# B&R Automation Studio project ShowCase2Mo410Test
Automation Studio 4.10.5.38 SP; technology packages: mapp 5.23.1, mappCockpit 5.23.0, mappMotion 5.23.1, mappView 5.23.0

## Configuration Config1

CPU X20CP1586, AutomationRuntime B4.91, Build 4.1.2, Safety 0.0, Vc 

### Task classes (Cpu.sw)
```
Cyclic#1:
  BoxLift <- BoxLift.prg
  ComTCP_P <- Libraries.ComTCP.ComTCP_P.prg
  AlarmBlink <- AlarmBlink.prg
  Axis1ST <- Axis1ST.prg
Cyclic#4:
  RecipeMgmt <- RecipeMgmt.prg
  PowerON <- PowerON.prg
  CamAutomat <- CamAutomat.prg
  LDMPAccess <- LDMPAccess.prg
DataObjects: McAcpSys
NcDataObjects: Cam <- Cam.dob, McDriveLog
Binaries: TCData, mvLoader, TCLang, udbdef, arsvcreg, mCoWebSc, arflatprv, arcoal, McAcpDrv, McAcpSim, arconfig, asfw, ashwd, iomap, User, Role, sysconf, TC, ashwac, Config_3, Config_2, Config, Config_1, Settings
Libraries: MTBasics, brsystem, MTTypes, sys_lib, runtime, ComTCP_L, operator, astime, AsTCP, standard, AsArLog, AsBrStr, MpRecipe, MpBase, McBase, CoTrace, AsZip, FileIO, MpAxis, McAxis, McAcpAx, asieccon, arssl, asepl, powerlnk
```

### Hardware
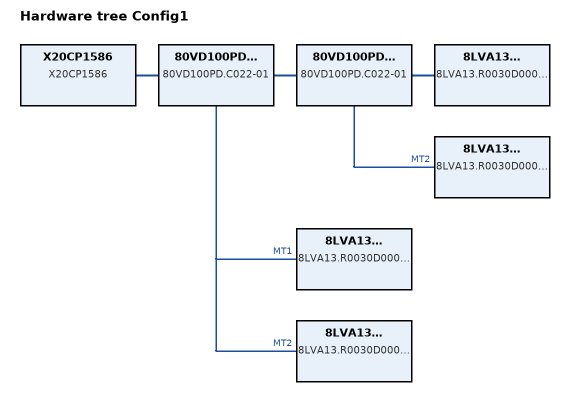
```
80VD100PD.C022-01 : 80VD100PD.C022-01 v2.5.0.0  [PLK1 -> X20CP1586.IF3 (NodeNumber=2) [Cable Type=PowerlinkCable, Length=10, Version=1.0.0.3]; PLK2 -> 80VD100PD.C022-01a.PLK1 (NodeNumber=2) [Cable Type=PowerlinkCable, Length=10, Version=1.0.0.3]; MT2 -> 8LVA13.R0030D000-0a.MT]
  DriveConfiguration/Module:
    McAcoposTypeID = AcoposMicroDConfig
    ActivateACOPOSSimulationOnPLC = 0
  DriveConfiguration/Encoder/EncoderX6A/InterfaceType:
    ResolverPolepairs = 1
  DriveConfiguration/Encoder/EncoderX6B/InterfaceType:
    ResolverPolepairs = 1
  DriveConfiguration/Channel[1]/RealAxis:
    AxisReference = gAxis3_MpLink
    MechanicalElementsIsInvisible = 0
  DriveConfiguration/Channel[1]/RealAxis/MechanicalElements/Gearbox:
    InputIsReadOnly = 0
    Input = 1
    OutputIsReadOnly = 0
    Output = 1
  DriveConfiguration/Channel[1]/RealAxis/MechanicalElements/RotaryToLinearTransformation:
    ReferenceDistanceIsReadOnly = 0
    ReferenceDistance = 1
  DriveConfiguration/Channel[1]/RealAxis/Controller:
    ModeIsReadOnly = 0
    Mode = PositionController
  DriveConfiguration/Channel[1]/RealAxis/Controller/Mode/Position:
    ProportionalGain = 50.0
    IntegrationTime = 0.0
    PredictionTime = 0.0004
    TotalDelayTime = 0.0004
  DriveConfiguration/Channel[1]/RealAxis/Controller/Mode/Speed:
    ProportionalGainIsReadOnly = 0
    ProportionalGain = 2.0
    IntegrationTimeIsReadOnly = 0
    IntegrationTime = 0.0
    FilterTimeIsReadOnly = 0
    FilterTime = 0.0
  DriveConfiguration/Channel[1]/RealAxis/Controller/Mode/LoopFilters:
    LoopFilterXIsReadOnly = 0
    LoopFilter1 = NotUsed
    LoopFilter2 = NotUsed
    LoopFilter3 = NotUsed
  DriveConfiguration/Channel[1]/RealAxis/Homing:
    ModeIsReadOnly = 0
    Mode = Direct
  DriveConfiguration/Channel[1]/RealAxis/Homing/Mode:
    Position = 0.0
    ReferencePulse = NotUsed
  DriveConfiguration/Channel[1]/RealAxis/Homing:
    RestorePositionVariable = 
  DriveConfiguration/Channel[1]/RealAxis/StopReaction:
    QuickstopIsReadOnly = 0
    Quickstop = DecelerationLimit
    DriveErrorIsReadOnly = 0
    DriveError = DecelerationLimit
  DriveConfiguration/Channel[1]/RealAxis/MovementErrorLimits:
    PositionError = 300
    VelocityErrorMonitoring = Automatic1
  DriveConfiguration/Channel[1]/RealAxis:
    JerkFilterIsReadOnly = 0
    JerkFilter = NotUsed
    ZeroVibrationFilter = NotUsed
  DriveConfiguration/Channel[1]/RealAxis/DigitalInputs/HomingSwitch:
    SourceIsReadOnly = 0
    Source = NotUsed
    Level = High
  DriveConfiguration/Channel[1]/RealAxis/DigitalInputs/PositiveLimitSwitch:
    SourceIsReadOnly = 0
    Source = NotUsed
    Level = High
  DriveConfiguration/Channel[1]/RealAxis/DigitalInputs/NegativeLimitSwitch:
    SourceIsReadOnly = 0
    Source = NotUsed
    Level = High
  DriveConfiguration/Channel[1]/RealAxis/DigitalInputs/Trigger1:
    Source = X2Trigger1
    Level = High
  DriveConfiguration/Channel[1]/RealAxis/DigitalInputs/Trigger2:
    Source = X2Trigger2
    Level = High
  DriveConfiguration/Channel[1]/RealAxis/DigitalInputs/Quickstop:
    Input = NotUsed
  DriveConfiguration/Channel[1]/RealAxis/Simulation:
    SimulationModeOnPLC = SetValueGeneration
    SimulationModeOnACOPOS = NotUsed
  DriveConfiguration/Channel[1]/RealAxis/AxisFeatures:
    FeatureRef[1] = 
  DriveConfiguration/Channel[1]:
    VirtualAxis = Used
  DriveConfiguration/Channel[1]/VirtualAxis:
    AxisReference = gAxisV3_MpLink
  DriveConfiguration/Channel[1]/VirtualAxis/Homing:
    Mode = Direct
  DriveConfiguration/Channel[1]/VirtualAxis/Homing/Mode:
    Position = 0.0
  DriveConfiguration/Channel[1]/VirtualAxis/Homing:
    RestorePositionVariable = 
  DriveConfiguration/Channel[1]/VirtualAxis:
    JerkFilterIsReadOnly = 0
    JerkFilter = NotUsed
    ZeroVibrationFilter = NotUsed
  DriveConfiguration/Channel[1]/ChannelFeatures:
    FeatureRef[1] = Feature_CamList
  DriveConfiguration/Channel[2]/RealAxis:
    AxisReference = gAxis4_MpLink
    MechanicalElementsIsInvisible = 0
  DriveConfiguration/Channel[2]/RealAxis/MechanicalElements/Gearbox:
    InputIsReadOnly = 0
    Input = 1
    OutputIsReadOnly = 0
    Output = 1
  DriveConfiguration/Channel[2]/RealAxis/MechanicalElements/RotaryToLinearTransformation:
    ReferenceDistanceIsReadOnly = 0
    ReferenceDistance = 1
  DriveConfiguration/Channel[2]/RealAxis/Controller:
    ModeIsReadOnly = 0
    Mode = PositionController
  DriveConfiguration/Channel[2]/RealAxis/Controller/Mode/Position:
    ProportionalGain = 50.0
    IntegrationTime = 0.0
    PredictionTime = 0.0004
    TotalDelayTime = 0.0004
  DriveConfiguration/Channel[2]/RealAxis/Controller/Mode/Speed:
    ProportionalGainIsReadOnly = 0
    ProportionalGain = 2.0
    IntegrationTimeIsReadOnly = 0
    IntegrationTime = 0.0
    FilterTimeIsReadOnly = 0
    FilterTime = 0.0
  DriveConfiguration/Channel[2]/RealAxis/Controller/Mode/LoopFilters:
    LoopFilterXIsReadOnly = 0
    LoopFilter1 = NotUsed
    LoopFilter2 = NotUsed
    LoopFilter3 = NotUsed
  DriveConfiguration/Channel[2]/RealAxis/Homing:
    ModeIsReadOnly = 0
    Mode = Direct
  DriveConfiguration/Channel[2]/RealAxis/Homing/Mode:
    Position = 0.0
    ReferencePulse = NotUsed
  DriveConfiguration/Channel[2]/RealAxis/Homing:
    RestorePositionVariable = 
  DriveConfiguration/Channel[2]/RealAxis/StopReaction:
    QuickstopIsReadOnly = 0
    Quickstop = DecelerationLimit
    DriveErrorIsReadOnly = 0
    DriveError = DecelerationLimit
  DriveConfiguration/Channel[2]/RealAxis/MovementErrorLimits:
    PositionError = 300
    VelocityErrorMonitoring = Automatic1
  DriveConfiguration/Channel[2]/RealAxis:
    JerkFilterIsReadOnly = 0
    JerkFilter = NotUsed
    ZeroVibrationFilter = NotUsed
  DriveConfiguration/Channel[2]/RealAxis/DigitalInputs/HomingSwitch:
    SourceIsReadOnly = 0
    Source = NotUsed
    Level = High
  DriveConfiguration/Channel[2]/RealAxis/DigitalInputs/PositiveLimitSwitch:
    SourceIsReadOnly = 0
    Source = NotUsed
    Level = High
  DriveConfiguration/Channel[2]/RealAxis/DigitalInputs/NegativeLimitSwitch:
    SourceIsReadOnly = 0
    Source = NotUsed
    Level = High
  DriveConfiguration/Channel[2]/RealAxis/DigitalInputs/Trigger1:
    Source = X2Trigger1
    Level = High
  DriveConfiguration/Channel[2]/RealAxis/DigitalInputs/Trigger2:
    Source = X2Trigger2
    Level = High
  DriveConfiguration/Channel[2]/RealAxis/DigitalInputs/Quickstop:
    Input = NotUsed
  DriveConfiguration/Channel[2]/RealAxis/Simulation:
    SimulationModeOnPLC = SetValueGeneration
    SimulationModeOnACOPOS = NotUsed
80VD100PD.C022-01a : 80VD100PD.C022-01 v2.5.0.0  [PLK1 -> 80VD100PD.C022-01.PLK2 (NodeNumber=1) [Cable Type=PowerlinkCable, Length=10, Version=1.0.0.3]; MT2 -> 8LVA13.R0030D000-0c.MT]
  DriveConfiguration/Module:
    McAcoposTypeID = AcoposMicroDConfig
    ActivateACOPOSSimulationOnPLC = 0
  DriveConfiguration/Encoder/EncoderX6A/InterfaceType:
    ResolverPolepairs = 1
  DriveConfiguration/Encoder/EncoderX6B/InterfaceType:
    ResolverPolepairs = 1
  DriveConfiguration/Channel[1]/RealAxis:
    AxisReference = gAxis1_MpLink
    MechanicalElementsIsInvisible = 0
  DriveConfiguration/Channel[1]/RealAxis/MechanicalElements/Gearbox:
    InputIsReadOnly = 0
    Input = 1
    OutputIsReadOnly = 0
    Output = 1
  DriveConfiguration/Channel[1]/RealAxis/MechanicalElements/RotaryToLinearTransformation:
    ReferenceDistanceIsReadOnly = 0
    ReferenceDistance = 1
  DriveConfiguration/Channel[1]/RealAxis/Controller:
    ModeIsReadOnly = 0
    Mode = PositionController
  DriveConfiguration/Channel[1]/RealAxis/Controller/Mode/Position:
    ProportionalGain = 50.0
    IntegrationTime = 0.0
    PredictionTime = 0.0004
    TotalDelayTime = 0.0004
  DriveConfiguration/Channel[1]/RealAxis/Controller/Mode/Speed:
    ProportionalGainIsReadOnly = 0
    ProportionalGain = 2.0
    IntegrationTimeIsReadOnly = 0
    IntegrationTime = 0.0
    FilterTimeIsReadOnly = 0
    FilterTime = 0.0
  DriveConfiguration/Channel[1]/RealAxis/Controller/Mode/LoopFilters:
    LoopFilterXIsReadOnly = 0
    LoopFilter1 = NotUsed
    LoopFilter2 = NotUsed
    LoopFilter3 = NotUsed
  DriveConfiguration/Channel[1]/RealAxis/Homing:
    ModeIsReadOnly = 0
    Mode = Direct
  DriveConfiguration/Channel[1]/RealAxis/Homing/Mode:
    Position = 0.0
    ReferencePulse = NotUsed
  DriveConfiguration/Channel[1]/RealAxis/Homing:
    RestorePositionVariable = 
  DriveConfiguration/Channel[1]/RealAxis/StopReaction:
    QuickstopIsReadOnly = 0
    Quickstop = DecelerationLimit
    DriveErrorIsReadOnly = 0
    DriveError = DecelerationLimit
  DriveConfiguration/Channel[1]/RealAxis/MovementErrorLimits:
    PositionError = 300
    VelocityErrorMonitoring = Automatic1
  DriveConfiguration/Channel[1]/RealAxis:
    JerkFilterIsReadOnly = 0
    JerkFilter = NotUsed
    ZeroVibrationFilter = NotUsed
  DriveConfiguration/Channel[1]/RealAxis/DigitalInputs/HomingSwitch:
    SourceIsReadOnly = 0
    Source = NotUsed
    Level = High
  DriveConfiguration/Channel[1]/RealAxis/DigitalInputs/PositiveLimitSwitch:
    SourceIsReadOnly = 0
    Source = NotUsed
    Level = High
  DriveConfiguration/Channel[1]/RealAxis/DigitalInputs/NegativeLimitSwitch:
    SourceIsReadOnly = 0
    Source = NotUsed
    Level = High
  DriveConfiguration/Channel[1]/RealAxis/DigitalInputs/Trigger1:
    Source = X2Trigger1
    Level = High
  DriveConfiguration/Channel[1]/RealAxis/DigitalInputs/Trigger2:
    Source = X2Trigger2
    Level = High
  DriveConfiguration/Channel[1]/RealAxis/DigitalInputs/Quickstop:
    Input = NotUsed
  DriveConfiguration/Channel[1]/RealAxis/Simulation:
    SimulationModeOnPLC = SetValueGeneration
    SimulationModeOnACOPOS = NotUsed
  DriveConfiguration/Channel[1]/RealAxis/AxisFeatures:
    FeatureRef[1] = 
  DriveConfiguration/Channel[1]:
    VirtualAxis = Used
  DriveConfiguration/Channel[1]/VirtualAxis:
    AxisReference = gAxisV_MpLink
  DriveConfiguration/Channel[1]/VirtualAxis/Homing:
    Mode = Direct
  DriveConfiguration/Channel[1]/VirtualAxis/Homing/Mode:
    Position = 0.0
  DriveConfiguration/Channel[1]/VirtualAxis/Homing:
    RestorePositionVariable = 
  DriveConfiguration/Channel[1]/VirtualAxis:
    JerkFilterIsReadOnly = 0
    JerkFilter = NotUsed
    ZeroVibrationFilter = NotUsed
  DriveConfiguration/Channel[1]/ChannelFeatures:
    FeatureRef[1] = Feature_CamList
  DriveConfiguration/Channel[2]/RealAxis:
    AxisReference = gAxis2_MpLink
    MechanicalElementsIsInvisible = 0
  DriveConfiguration/Channel[2]/RealAxis/MechanicalElements/Gearbox:
    InputIsReadOnly = 0
    Input = 1
    OutputIsReadOnly = 0
    Output = 1
  DriveConfiguration/Channel[2]/RealAxis/MechanicalElements/RotaryToLinearTransformation:
    ReferenceDistanceIsReadOnly = 0
    ReferenceDistance = 1
  DriveConfiguration/Channel[2]/RealAxis/Controller:
    ModeIsReadOnly = 0
    Mode = PositionController
  DriveConfiguration/Channel[2]/RealAxis/Controller/Mode/Position:
    ProportionalGain = 50.0
    IntegrationTime = 0.0
    PredictionTime = 0.0004
    TotalDelayTime = 0.0004
  DriveConfiguration/Channel[2]/RealAxis/Controller/Mode/Speed:
    ProportionalGainIsReadOnly = 0
    ProportionalGain = 2.0
    IntegrationTimeIsReadOnly = 0
    IntegrationTime = 0.0
    FilterTimeIsReadOnly = 0
    FilterTime = 0.0
  DriveConfiguration/Channel[2]/RealAxis/Controller/Mode/LoopFilters:
    LoopFilterXIsReadOnly = 0
    LoopFilter1 = NotUsed
    LoopFilter2 = NotUsed
    LoopFilter3 = NotUsed
  DriveConfiguration/Channel[2]/RealAxis/Homing:
    ModeIsReadOnly = 0
    Mode = Direct
  DriveConfiguration/Channel[2]/RealAxis/Homing/Mode:
    Position = 0.0
    ReferencePulse = NotUsed
  DriveConfiguration/Channel[2]/RealAxis/Homing:
    RestorePositionVariable = 
  DriveConfiguration/Channel[2]/RealAxis/StopReaction:
    QuickstopIsReadOnly = 0
    Quickstop = DecelerationLimit
    DriveErrorIsReadOnly = 0
    DriveError = DecelerationLimit
  DriveConfiguration/Channel[2]/RealAxis/MovementErrorLimits:
    PositionError = 300
    VelocityErrorMonitoring = Automatic1
  DriveConfiguration/Channel[2]/RealAxis:
    JerkFilterIsReadOnly = 0
    JerkFilter = NotUsed
    ZeroVibrationFilter = NotUsed
  DriveConfiguration/Channel[2]/RealAxis/DigitalInputs/HomingSwitch:
    SourceIsReadOnly = 0
    Source = NotUsed
    Level = High
  DriveConfiguration/Channel[2]/RealAxis/DigitalInputs/PositiveLimitSwitch:
    SourceIsReadOnly = 0
    Source = NotUsed
    Level = High
  DriveConfiguration/Channel[2]/RealAxis/DigitalInputs/NegativeLimitSwitch:
    SourceIsReadOnly = 0
    Source = NotUsed
    Level = High
  DriveConfiguration/Channel[2]/RealAxis/DigitalInputs/Trigger1:
    Source = X2Trigger1
    Level = High
  DriveConfiguration/Channel[2]/RealAxis/DigitalInputs/Trigger2:
    Source = X2Trigger2
    Level = High
  DriveConfiguration/Channel[2]/RealAxis/DigitalInputs/Quickstop:
    Input = NotUsed
  DriveConfiguration/Channel[2]/RealAxis/Simulation:
    SimulationModeOnPLC = SetValueGeneration
    SimulationModeOnACOPOS = NotUsed
8LVA13.R0030D000-0 : 8LVA13.R0030D000-0 v2.2.0.3  [MT -> 80VD100PD.C022-01.MT1]
  M1/MotorParameters:
    MOTOR_AMB_TEMP_RATED = 40
8LVA13.R0030D000-0a : 8LVA13.R0030D000-0 v2.2.0.3  [MT -> 80VD100PD.C022-01.MT2]
  M1/MotorParameters:
    MOTOR_AMB_TEMP_RATED = 40
8LVA13.R0030D000-0b : 8LVA13.R0030D000-0 v2.2.0.3  [MT -> 80VD100PD.C022-01a.MT1]
  M1/MotorParameters:
    MOTOR_AMB_TEMP_RATED = 40
8LVA13.R0030D000-0c : 8LVA13.R0030D000-0 v2.2.0.3  [MT -> 80VD100PD.C022-01a.MT2]
  M1/MotorParameters:
    MOTOR_AMB_TEMP_RATED = 40
X20CP1586 : X20CP1586 v1.9.0.0
  Connector IF2:
    ActivateDevice = 1
    HostName = mo
    Mode = Manual
    InternetAddress = 192.168.2.32
    SubnetMask = 255.255.255.0
  Connector IF3:
    DNAConfiguration = manual
  ConfigurationID = mappViewGettingStarted_ETA210_T50
  UserPartitionSize = 200
  Simulation = 1
  FileDevice1
  FileDeviceName1 = CSV_Recipes
  FileDevicePath1 = F:\Recipes
  FileDevice2
  FileDeviceName2 = SIM_Recipes
  FileDevicePath2 = C:\Basic
  FtpUser1
  FtpUsername1 = academy
  FtpUserPassword1 = PTbbKbjlQWNQQLeLnvYxsprPr7USEpMWmZovrSfugvI=
  FtpUserSalt1 = LwThsYzd
  FTPAccessRight1 = 0
  ActivateOpcUa = 1
  OpcUaInformationModels_PV_Version = 1
```

### PvMap.vvm - X20CP1586/PvMap.vvm
```iecst
VAR_CONFIG
	::ComTCP_SimActive AT %Q.::gComTCPSimActive; (*Insert your comment here...*)
	::BoxLift:aoBottomBoxReleaseTime AT %Q.::ComTCP_SimOutputs.BottomBox_ReleaseTime; (*Insert your comment here...*)
	::BoxLift:aoTopBoxReleaseTime AT %Q.::ComTCP_SimOutputs.TopBox_ReleaseTime; (*Insert your comment here...*)
	::ComTCP_SimInputs.diConvTop AT %Q.::BoxLift:diConvTop; (*Insert your comment here...*)
	::ComTCP_SimInputs.diConvBottom AT %Q.::BoxLift:diConvBottom; (*Insert your comment here...*)
	::ComTCP_SimInputs.diBoxLift AT %Q.::BoxLift:diBoxLift; (*Insert your comment here...*)
	::ComTCP_SimInputs.diUnloaded AT %Q.::BoxLift:diUnloaded; (*Insert your comment here...*)
	::ComTCP_SimInputs.diLiftTop AT %Q.::BoxLift:diLiftTop; (*Insert your comment here...*)
	::ComTCP_SimInputs.diLiftBottom AT %Q.::BoxLift:diLiftBottom; (*Insert your comment here...*)
	::ComTCP_SimInputs.diLiftUnload AT %Q.::BoxLift:diLiftUnload; (*Insert your comment here...*)
	::BoxLift:doConvTop AT %Q.::ComTCP_SimOutputs.doConvTop; (*Insert your comment here...*)
	::BoxLift:doConvBottom AT %Q.::ComTCP_SimOutputs.doConvBottom; (*Insert your comment here...*)
	::BoxLift:doConvLift AT %Q.::ComTCP_SimOutputs.doConvLift; (*Insert your comment here...*)
	::BoxLift:doLiftTop AT %Q.::ComTCP_SimOutputs.doLiftTop; (*Insert your comment here...*)
	::BoxLift:doLiftBottom AT %Q.::ComTCP_SimOutputs.doLiftBottom; (*Insert your comment here...*)
	::BoxLift:doLiftUnload AT %Q.::ComTCP_SimOutputs.doLiftUnload; (*Insert your comment here...*)
	::BoxLift:aoConvBottomVelocity AT %Q.::ComTCP_SimOutputs.ConvBottom_Velocity; (*Insert your comment here...*)
	::BoxLift:aoConvLiftVelocity AT %Q.::ComTCP_SimOutputs.ConvLift_Velocity; (*Insert your comment here...*)
	::BoxLift:aoConvTopVelocity AT %Q.::ComTCP_SimOutputs.ConvTop_Velocity; (*Insert your comment here...*)
	::BoxLift:aoInfeedConvBottomVelocity AT %Q.::ComTCP_SimOutputs.InfeedConvBottom_Velocity; (*Insert your comment here...*)
	::BoxLift:aoInfeedConvTopVelocity AT %Q.::ComTCP_SimOutputs.InfeedConvTop_Velocity; (*Insert your comment here...*)
	::BoxLift:aoOutfeedConvVelocity AT %Q.::ComTCP_SimOutputs.OutfeedConv_Velocity; (*Insert your comment here...*)
END_VAR
```

### Config_1.axis - X20CP1586/mappMotion/Config_1.axis
```
Element gAxis2_MpLink (Type=axis)  // Axis 2 not used
  BaseTypeIsReadOnly = 0
  BaseType = Linear
    MeasurementUnit = 5066068
    MeasurementResolutionIsReadOnly = 0
    MeasurementResolution = 0.01
    CountDirectionIsReadOnly = 0
    CountDirection = Standard
  MovementLimitsIsReadOnly = 0
  MovementLimits = Internal
    Position:
      LowerLimitMin = -1.79769313486231E308
      UpperLimitMax = 1.79769313486231E308
      LowerLimit = -1000.0
      UpperLimit = 1000.0
    VelocityIsReadOnly = 0
    Velocity:
      VelocityMax = 3.4E38
      Velocity = 15000
    AccelerationIsReadOnly = 0
    Acceleration:
      AccelerationMax = 3.4E38
      Acceleration = 150000
    DecelerationIsReadOnly = 0
    Deceleration:
      DecelerationMax = 3.4E38
      Deceleration = 150000
  Alarms = MpAlarmX
Element gAxisV3_MpLink (Type=axis)  // Virtual axis for servo 3
  BaseTypeIsReadOnly = 0
  BaseType = Linear
    MeasurementUnit = 5066068
    MeasurementResolutionIsReadOnly = 0
    MeasurementResolution = 0.01
    CountDirectionIsReadOnly = 0
    CountDirection = Standard
  MovementLimitsIsReadOnly = 0
  MovementLimits = Internal
    Position:
      LowerLimitMin = -1.79769313486231E308
      UpperLimitMax = 1.79769313486231E308
      LowerLimit = -1000.0
      UpperLimit = 1000.0
    VelocityIsReadOnly = 0
    Velocity:
      VelocityMax = 3.4E38
      Velocity = 15000
    AccelerationIsReadOnly = 0
    Acceleration:
      AccelerationMax = 3.4E38
      Acceleration = 150000
    DecelerationIsReadOnly = 0
    Deceleration:
      DecelerationMax = 3.4E38
      Deceleration = 150000
  Alarms = MpAlarmX
Element gAxisV_MpLink (Type=axis)  // Virtual axis for servo 1
  BaseTypeIsReadOnly = 0
  BaseType = Linear
    MeasurementUnit = 5066068
    MeasurementResolutionIsReadOnly = 0
    MeasurementResolution = 0.01
    CountDirectionIsReadOnly = 0
    CountDirection = Standard
  MovementLimitsIsReadOnly = 0
  MovementLimits = Internal
    Position:
      LowerLimitMin = -1.79769313486231E308
      UpperLimitMax = 1.79769313486231E308
      LowerLimit = -1000.0
      UpperLimit = 1000.0
    VelocityIsReadOnly = 0
    Velocity:
      VelocityMax = 3.4E38
      Velocity = 15000
    AccelerationIsReadOnly = 0
    Acceleration:
      AccelerationMax = 3.4E38
      Acceleration = 150000
    DecelerationIsReadOnly = 0
    Deceleration:
      DecelerationMax = 3.4E38
      Deceleration = 150000
  Alarms = MpAlarmX
Element gAxis4_MpLink (Type=axis)  // Axis 4 not used
  BaseTypeIsReadOnly = 0
  BaseType = Linear
    MeasurementUnit = 5066068
    MeasurementResolutionIsReadOnly = 0
    MeasurementResolution = 0.01
    CountDirectionIsReadOnly = 0
    CountDirection = Standard
  MovementLimitsIsReadOnly = 0
  MovementLimits = Internal
    Position:
      LowerLimitMin = -1.79769313486231E308
      UpperLimitMax = 1.79769313486231E308
      LowerLimit = -1000.0
      UpperLimit = 1000.0
    VelocityIsReadOnly = 0
    Velocity:
      VelocityMax = 3.4E38
      Velocity = 15000
    AccelerationIsReadOnly = 0
    Acceleration:
      AccelerationMax = 3.4E38
      Acceleration = 150000
    DecelerationIsReadOnly = 0
    Deceleration:
      DecelerationMax = 3.4E38
      Deceleration = 150000
  Alarms = MpAlarmX
Element gAxis3_MpLink (Type=axis)  // Axis 3 the lift conveyor with cam automat
  BaseTypeIsReadOnly = 0
  BaseType = Linear
    MeasurementUnit = 5066068
    MeasurementResolutionIsReadOnly = 0
    MeasurementResolution = 0.01
    CountDirectionIsReadOnly = 0
    CountDirection = Standard
  MovementLimitsIsReadOnly = 0
  MovementLimits = Internal
    Position:
      LowerLimitMin = -1.79769313486231E308
      UpperLimitMax = 1.79769313486231E308
      LowerLimit = -1000.0
      UpperLimit = 1000.0
    VelocityIsReadOnly = 0
    Velocity:
      VelocityMax = 3.4E38
      Velocity = 15000
    AccelerationIsReadOnly = 0
    Acceleration:
      AccelerationMax = 3.4E38
      Acceleration = 150000
    DecelerationIsReadOnly = 0
    Deceleration:
      DecelerationMax = 3.4E38
      Deceleration = 150000
  Alarms = MpAlarmX
Element gAxis1_MpLink (Type=axis)  // Axis 1 the lift conveyor
  BaseTypeIsReadOnly = 0
  BaseType = Linear
    MeasurementUnit = 5066068
    MeasurementResolutionIsReadOnly = 0
    MeasurementResolution = 0.01
    CountDirectionIsReadOnly = 0
    CountDirection = Standard
  MovementLimitsIsReadOnly = 0
  MovementLimits = Internal
    Position:
      LowerLimitMin = -1.79769313486231E308
      UpperLimitMax = 1.79769313486231E308
      LowerLimit = -1000.0
      UpperLimit = 1000.0
    VelocityIsReadOnly = 0
    Velocity:
      VelocityMax = 3.4E38
      Velocity = 15000
    AccelerationIsReadOnly = 0
    Acceleration:
      AccelerationMax = 3.4E38
      Acceleration = 150000
    DecelerationIsReadOnly = 0
    Deceleration:
      DecelerationMax = 3.4E38
      Deceleration = 150000
  Alarms = MpAlarmX
```

### Config_3.axisfeature - X20CP1586/mappMotion/Config_3.axisfeature
```
Element Feature_CamList_3 (Type=axisfeature)
  Type = CamList
    CamListRef = CamList_3
Element Feature_CamList (Type=axisfeature)
  Type = CamList
    CamListRef = CamList_1
```

### Config_4.camlist - X20CP1586/mappMotion/Config_4.camlist
```
Element CamList_3 (Type=camlist)
  Row[1]:
    CamName = Cam3
    CamID = 3
    Description
```

## Logical view

Binary libraries used (declarations not repeated): operator, runtime, astime, AsIecCon, brsystem, sys_lib, AsTCP, standard, AsArLog, AsBrStr, MpRecipe, MpBase, McBase, MTBasics 5.12.0, MTTypes, CoTrace, AsZip, FileIO, MpAxis, McAxis, McAcpAx

### Global.typ - Global data types
```iecst
TYPE
	iPhysicParam_typ : 	STRUCT
		UserOutfeedConvVelocity : REAL := 1.0; (*OutfeedConv Velocity Speed ref*)
		UserInfeedConvTopVelocity : REAL := 0.6; (* InfeedConvTop Velocity Speed ref*)
		UserInfeedConvBottomVelocity : REAL := 0.5; (*InfeedConvBottom Velocity Speed ref*)
		UserConvTopVelocity : REAL := 1.0; (* ConvTop VelocitySpeed ref*)
		UserConvLiftVelocity : REAL := 1.0; (* ConvLift Velocity Speed ref*)
		UserConvBottomVelocity : REAL := 1.0; (* Conv Bottom Velocity Speed ref*)
		UserTopBoxReleaseTime : REAL := 25.0;
		UserBottomBoxReleaseTime : REAL := 20.0;
		BlockSensorLowerConvTime : TIME := T#500ms;
		BlockSensorUpperConvTime : TIME := T#500ms;
		MaximumUloadedBox : REAL := 0.0; (*Maximum unloaded box at each speed*)
	END_STRUCT;
	Axis_type : 	STRUCT
		Exists : BOOL;
		name : STRING[10]; (*Name of the axis*)
		cmdReset : BOOL; (*cmd from HMI to reset any fault*)
		cmdStart : BOOL; (*cmd to start this axis *)
		cmdCam : BOOL;
		cmdGear : BOOL;
		cmdStop : BOOL; (*cmd to stop this axis*)
		cmdHome : BOOL; (*cmd from HMI to home this axis*)
		cmdReference : BOOL; (*cmd from HMI to set the zero offset of the axis.*)
		cmdRun : BOOL; (*cmd to put axis into run state*)
		cmdOffset : BOOL;
		cmdJog : BOOL; (*cmd to put axis into jog state*)
		cmdManualForward : BOOL; (*cmd from HMI to put axis into manual forward state*)
		cmdManualReverse : BOOL; (*cmd from HMI to put axis into manual reverse state*)
		cmdMoveAbsolute : BOOL; (*cmd from control task to move axis to absolute position*)
		parmSpeed : REAL; (*cmded speed for manual moves*)
		parmAccelDecel : REAL; (*Acceleration and deceleration of absolute moves*)
		parmAbsolutePosition : REAL; (*Absolute position for absolute moves*)
		parmMaxTorque : REAL; (*Max torque when torque limiting is enabled*)
		statusOn : BOOL; (*Axis is powered on*)
		statusOff : BOOL; (*Axis is powered off*)
		statusDisabled : BOOL; (*Hardware disabled*)
		statusFaulted : BOOL; (*Axis is in the Faulted State*)
		statusStarting : BOOL; (*Axis is in the Starting State*)
		statusHoming : BOOL; (*Axis is in the Homing State*)
		statusInPosition : BOOL; (*Axis is in position following an absolute move*)
		statusRunning : BOOL; (*Axis is in the Running State*)
		statusJogging : BOOL; (*Axis is in the Jogging State*)
		statusMoving : BOOL; (*Axis velocity is > 0*)
		statusManualForward : BOOL; (*Axis is in the Manual Forward State*)
		statusManualReverse : BOOL; (*Axis is in the Manual Reverse State*)
		statusStopping : BOOL; (*Axis is in the Manual Stopping State*)
		statusHomed : BOOL; (*Axis has been homed*)
		statusPosition : LREAL; (*Axis position*)
		statusSpeed : REAL; (*Axis speed*)
		statusCurrent : REAL; (*Axis motor current *)
		statusLagError : REAL; (*Axis lag error*)
		statusTemperature : REAL; (*Actual Temperature*)
		statusTorque : REAL; (*Actual Torque*)
		statusMasterOffset : LREAL; (*Actual offset from master*)
		statusAbsMoveActive : BOOL; (*Absolute move is active*)
		statusGeared : BOOL; (*Axis is geared with the master*)
		statusPoweredOff : BOOL; (*Axis is powered OFF from the software*)
		statusStopped : BOOL; (*Axis has stopped moving*)
		statusPeakCurrent : REAL; (*Peak over the last few seconds motor current *)
		statusPeakLagError : REAL; (*Peak over the last few seconds lag error*)
		statusPeakTorque : REAL; (*Peak over the last few seconds Torque*)
		statusErrorID : UDINT; (*Axis ErrorID (0=no error)*)
		parmMaintMax : REAL;
		parmMaintMin : REAL;
		parmMax : REAL; (*Position to move to when cmded to park. (Real world units)*)
		parmMin : REAL; (*Position to move to when cmded to park. (Real world units)*)
		parmOperMax : REAL; (*Max position displayed on screen based on job setup and mechanical limits*)
		parmOperMin : REAL; (*Min position displayed on screen based on job setup and mechanical limits*)
		parmReferencePosition : REAL; (*Physical position when at the reference mark. (Real world units)*)
	END_STRUCT;
END_TYPE
```

### Global.var - Global variables
```iecst
VAR
	gActivateMotion : BOOL;
	gComTCPSimActive : BOOL;
	gDispalyAlarm : BOOL; (*Dispaly Alarm*)
	gDispalyNoComm : BOOL; (*Display Stop image*)
	gDispalyRun : BOOL; (*dispaly Run image*)
	gDispalyStop : BOOL; (*Display Stop image*)
	gDisplayBlink : BOOL;
	gSaveParameter : BOOL;
END_VAR
VAR RETAIN
	gSiPhysics : ARRAY[0..2] OF iPhysicParam_typ;
	gSpeedRefHmi : INT;
END_VAR
VAR
	gUserReset : BOOL; (*User input to reset errors*)
	gUserStart : BOOL; (*User start input*)
	gUserStop : BOOL; (*User start input*)
	gReceiptChanged : BOOL;
END_VAR
VAR RETAIN
	gErrorDes : ARRAY[0..9] OF STRING[80];
	gErrorTime : ARRAY[0..9] OF DATE_AND_TIME;
	gBoxCountUnload : CTU;
END_VAR
VAR
	Axis3 : Axis_type := (Exists:=1);
	Axis1 : Axis_type := (Exists:=1);
	gAxisPosition : ARRAY[0..1] OF REAL;
	gMpAxisBasic_Axis2 : MpAxisBasic;
	gMpAxisBasic_Axis1 : MpAxisBasic;
	gMpAxisBasic_AxisVirtu : MpAxisBasic;
	gMpAxisCoupling_0 : MpAxisCoupling;
	gMpAxisBasicParType_Axis2 : MpAxisBasicParType;
	gMpAxisBasicParType_AxisVirtu : MpAxisBasicParType;
	gMpAxisBasicParType_Axis1 : MpAxisBasicParType;
	gCouplingPar : MpAxisCouplingParType;
	gMpAxisBasic_Axis4 : MpAxisBasic;
	gMpAxisBasic_Axis3 : MpAxisBasic;
	gMpAxisBasic_AxisVirtu3 : MpAxisBasic;
	gMpAxisCoupling_3 : MpAxisCoupling;
	gMpAxisBasicParType_Axis4 : MpAxisBasicParType;
	gMpAxisBasicParType_AxisVirtu3 : MpAxisBasicParType;
	gMpAxisBasicParType_Axis3 : MpAxisBasicParType;
	gCouplingPar3 : MpAxisCouplingParType;
	userRatioDenominator : UINT;
	userRatioNumerator : UINT;
	gServoInitialized : BOOL;
	gSpeedFactor : REAL := 1.0;
END_VAR
```

### Package Logical/Libraries - Global libraries

- Visualisation Logical/mappView (not shown)

### Program Logical/BoxLift (IEC) - Main Program Control Alarm

#### Types.typ
```iecst
TYPE
	State_enum :
		( (*State of the box lift*)
		STOP := 0,
		MAKE := 1,
		UNLOAD := 2,
		LOWER := 3,
		UPPER := 4,
		ERROR := 5,
		INIT := 6
		);
END_TYPE
```

#### Variables.var
```iecst
VAR
	aoBottomBoxReleaseTime : REAL;
	aoConvBottomVelocity : REAL; (*Conv Bottom Velocity Speed Control*)
	aoConvLiftVelocity : REAL; (*ConvLift Velocity Speed Control*)
	aoConvTopVelocity : REAL; (*ConvTop VelocitySpeed Control*)
	aoInfeedConvBottomVelocity : REAL; (*InfeedConvBottom Velocity Speed Control*)
	aoInfeedConvTopVelocity : REAL; (*InfeedConvTop Velocity Speed Control*)
	aoOutfeedConvVelocity : REAL; (*OutfeedConv Velocity Speed Control*)
	aoTopBoxReleaseTime : REAL;
	BoxCountUnloadDis : UINT;
	CopyDone : BOOL;
	CounterJamInfeed : CTU := (PV:=2);
	diBoxLift : BOOL; (*Box Detection at Lift*)
	diConvBottom : BOOL; (*Box Detection at Top conveyor*)
	diConvTop : BOOL; (*Box Detection at Top conveyor*)
	diLiftBottom : BOOL; (*Lift Bottom Position Feedback*)
	diLiftTop : BOOL; (*Lift Top Position Feedback*)
	diLiftUnload : BOOL; (*Lift Unload Position Feedback*)
	diUnloaded : BOOL; (*Unloaded Box off lift sensor*)
	doConvBottom : BOOL; (*Bottom Conveyor Run Cmd*)
	doConvLift : BOOL; (*Lift Conveyor Run Cmd*)
	doConvTop : BOOL; (*Top Conveyor Run Cmd*)
	doLiftBottom : BOOL; (*Lift Bottom Position Cmd*)
	doLiftTop : BOOL; (*Lift Top Position Cmd*)
	doLiftUnload : BOOL; (*Lift Unload Position Cmd*)
	DTGetTime_0 : DTGetTime;
END_VAR
VAR RETAIN
	ErrorDes : ARRAY[0..9] OF STRING[80];
END_VAR
VAR
	ErrorID : UDINT; (*0 = No Error. 1=Infeed Jam Lower  2=Infeed Jam Upper*)
	ErrorTable : ARRAY[0..10] OF STRING[80] := ['No Error','Lower Conveyor Error','Upper Conveyor Error','Uloading Error','Upper Conveyor Product Sensor Block','Lower Conveyor Product Sensor Block','Communication With iPhysics Error','Error Extra Box On Lift Conveyor',3('')];
	ErrorTimeString : ARRAY[0..9] OF STRING[80];
	i : UINT; (*memeory for shift alaram*)
	MemoUpperDischarge : BOOL; (*Will be on any time one lower picked up *)
	oneMinTimer : TON := (PT:=T#10s);
	Performance : UINT;
	PrevBoxCountUnload : UINT;
	ResetCount : BOOL;
	SaveAlarm : BOOL;
	SpeedInfoText : STRING[30];
	SpeedInfoTextTable : ARRAY[0..2] OF STRING[30] := ['Speed: Low','Speed: Medium','Speed: High']; (*For chart dispaly info*)
	State : State_enum;
	StatusDispaly : STRING[50];
	StatusDispalyDefault : ARRAY[0..9] OF STRING[50] := ['STOP','RUN - Wait For Box','RUN - Unloading Lower Conveyor','RUN - Unloading Upper Conveyor','RUN - Unloading Lift Conveyor','ERROR',4('')];
	StatusDispalyTopContent : STRING[50];
	StatusDispalyTopContentDefault : ARRAY[0..9] OF STRING[50] := ['Status: Stop',4('Status: Run'),'Status: Error','Status: Initializing Servos',3('')];
	TimerCommErrorIphysic : TON := (PT:=T#1500ms);
	TimerLowerSensorBlock : TON := (PT:=T#500ms);
	TimerUpperSensorBlock : TON := (PT:=T#500ms);
	TotalBoxUnloaded : UINT; (*Total box current job at 10s*)
	TotalBoxUnloadedPerSpeed : ARRAY[0..2] OF REAL; (*Total box unloaded at different speed at 10s*)
	UserBottomBoxReleaseTime : REAL := 20;
	UserConvBottomVelocity : REAL := 1.0; (*Conv Bottom Velocity Speed ref*)
	UserConvLiftVelocity : REAL := 1.0; (*ConvLift Velocity Speed ref*)
	UserConvTopVelocity : REAL := 1.0; (*ConvTop VelocitySpeed ref*)
	UserInfeedConvBottomVelocity : REAL := 0.5; (*InfeedConvBottom Velocity Speed ref*)
	UserInfeedConvTopVelocity : REAL := 0.6; (*InfeedConvTop Velocity Speed ref*)
	UserOutfeedConvVelocity : REAL := 1.0; (*OutfeedConv Velocity Speed ref*)
	UserTopBoxReleaseTime : REAL := 25;
	DispalyGraph : ARRAY[0..2] OF REAL := [1,2,3]; (*Graph info*)
	TotalBoxUnloadedPerSpeedLow : REAL;
	TotalBoxUnloadedPerSpeedMeduim : REAL;
	TotalBoxUnloadedPerSpeedHigh : REAL;
	diBoxLiftFilter : TON := (PT:=T#50ms); (*di Sensors noise filter*)
	diLiftTopFilter : TON := (PT:=T#50ms); (*di Sensors noise filter*)
	diLiftBottomFilter : TON := (PT:=T#50ms); (*di Sensors noise filter*)
	diConvBottomFilter : TON := (PT:=T#50ms);
	diConvTopFilter : TON := (PT:=T#50ms);
	diBoxLiftTON : TON := (PT:=T#350ms); (*Predict Boxon the lift conveyor*)
	BoxIsPassed : BOOL; (*Box Pass Memo*)
	Test_Bit_0 : BOOL; (*To be deleted just for test*)
END_VAR
```

#### Cyclic.st
```iecst
PROGRAM _CYCLIC

	CASE State OF

		STOP:  //***********************STOP**********************************************STOP********************************************STOP
			aoConvTopVelocity 			:= 0.0;   	// Turn off the Conv Top
			aoInfeedConvTopVelocity  	:= 0.0; 	// Turn off the Infeed Conv Top
			aoConvLiftVelocity 			:= 0.0; 	// Turn off the Conv Lift
			aoInfeedConvBottomVelocity 	:= 0.0; 	// Turn off the Infeed Conv Bottom
			aoOutfeedConvVelocity 		:= 0.0; 	// Turn off outfeed Conv
			aoConvBottomVelocity  		:= 0.0;   // Turn off the Conv Top
			aoTopBoxReleaseTime         := 100;  		//Box Release Speed
			aoBottomBoxReleaseTime      := 100; 	//Box Release Speed
			doLiftUnload 				:= FALSE; //Lift Unload Position Cmd
			doLiftTop 					:= FALSE; //Lift Top Position Cmd
			doLiftBottom 				:= FALSE; //Lift Bottom Position Cmd
			doConvTop 					:= FALSE; //Top Conveyor Run Cmd
			doConvLift 					:= FALSE; //Lift Conveyor Run Cmd
			doConvBottom 				:= FALSE; //Bottom Conveyor Run
			/// STOP Animation
			gDispalyStop 	:= TRUE; 	// Dispaly Stop Image
			gDispalyRun 	:= FALSE;   // Not Dispaly Run Image
			gDispalyAlarm 	:=FALSE;  	// Not Dispaly Alarm Image
			gUserStop 		:= FALSE;
			gUserReset 		:= FALSE;
			BoxIsPassed 	:= FALSE;
			i:=9;
			IF gUserStart THEN
				State := MAKE;
				gUserStart := FALSE;

			END_IF
			IF NOT gServoInitialized THEN
				State := INIT;

			END_IF

		MAKE:  //**************** MAKE *********************************************** MAKE ********************************************************************* MAKE

			/// RUN Animation
			gDispalyRun 		:= TRUE;    //Dispaly Run Image
			gDispalyStop		:= FALSE; 	// Dispaly Stop Image
			gDispalyAlarm 		:=FALSE;  	// Not Dispaly Alarm Image
			/// RUN Animation
			doConvTop    		:= NOT diConvTop;   	// Run the Top Conv
			doConvLift   		:= ( NOT diBoxLift OR BoxIsPassed);   	// Run the Lift Conv
			doConvBottom 		:= NOT diConvBottom; 	// Run the bottom conv

			CounterJamInfeed.RESET := TRUE;
			CounterJamInfeed();

			aoConvTopVelocity           := UserConvTopVelocity;   		// Set Speed the Conv Top
			aoConvBottomVelocity        := UserConvBottomVelocity;   	// Set Speed the Conv Top
			aoConvLiftVelocity          := UserConvLiftVelocity ; 		// Set Speed the Conv Lift
			aoOutfeedConvVelocity       := UserOutfeedConvVelocity; 	// Set Speed outfeed Conv
			aoInfeedConvTopVelocity     := UserInfeedConvTopVelocity ; 		// Set Speed the Infeed Conv Top
			aoInfeedConvBottomVelocity  := UserInfeedConvBottomVelocity; 	// Set Speed the Infeed Conv Bottom
			aoTopBoxReleaseTime         := UserTopBoxReleaseTime;  		//Box Release Speed
			aoBottomBoxReleaseTime      := UserBottomBoxReleaseTime; 	//Box Release Speed

			IF (diConvBottom AND NOT diConvTop AND NOT diBoxLift AND NOT BoxIsPassed ) THEN   // Sensor at the edge of the bottom conveyor detected with no box on the unload conv
				doConvBottom	:= FALSE; // Stop the bottom conv
				State 			:= LOWER;
			END_IF

			IF (diConvTop AND diConvBottom AND NOT MemoUpperDischarge AND NOT diBoxLift AND NOT BoxIsPassed) THEN   // Sensor at the edge of the bottom conveyor detected with no box on the unload conv Prio given to
				doConvTop    		:= FALSE;   // Stop the Top Conv
				MemoUpperDischarge 	:= TRUE;
				State := UPPER;
			ELSIF ( diConvTop AND diConvBottom AND MemoUpperDischarge AND NOT diBoxLift AND NOT BoxIsPassed)  THEN   // Sensor at the edge of the bottom conveyor detected with no box on the unload conv  Prio given to
				doConvBottom 		:= FALSE; // Stop the bottom conv
				MemoUpperDischarge 	:= FALSE;
				State := LOWER;
			END_IF

			IF (diConvTop AND NOT diConvBottom AND NOT diBoxLift AND NOT BoxIsPassed) THEN // Sensor at the edge of the top conveyor detected with no box on the unload conv
				doConvTop   := FALSE;   // Stop the Top Conv
				State 		:= UPPER;
			END_IF
			IF diBoxLift OR BoxIsPassed THEN  // Sensor at the center of the unload conveyor detected
				doConvLift  := BoxIsPassed;   // Stop the Lift Conv
				BoxIsPassed := FALSE;
				State 		:= UNLOAD;   // Change the state to UnLoad
			END_IF
			TimerCommErrorIphysic.IN := NOT gComTCPSimActive ;  // Detect communication Error iPhysic
			TimerCommErrorIphysic();
			IF TimerCommErrorIphysic.Q THEN //Infeed Jam Lower code
				ErrorID 		:= 6;  //Infeed Jam Lower Error
				State 			:= ERROR;
				gDispalyNoComm 	:= TRUE;
			END_IF

			IF gUserStop THEN
				gUserStop := FALSE;
				State := STOP;
			END_IF

		LOWER: //**************** LOWER *********************************************** LOWER ********************************************************************* LOWER

			doLiftBottom    := TRUE; //Move the lift conv to Bottom pos
			doConvTop    	:= NOT diConvTop ;   // Stop the Top Conv
			CounterJamInfeed.RESET 	:= FALSE;
			CounterJamInfeed.CU 	:= diConvBottomFilter.Q; // Count jammed box
			CounterJamInfeed();
			IF CounterJamInfeed.Q THEN
				ErrorID := 1;  //Infeed Jam Lower Error
				State 	:= ERROR;
			END_IF

			TimerLowerSensorBlock.IN := diConvBottom AND doConvBottom ;  // Detect sensor block if the conv run
			TimerLowerSensorBlock();

			IF TimerLowerSensorBlock.Q THEN //Infeed Jam Lower code
				ErrorID := 5;  //Infeed Jam Lower Error
				State 	:= ERROR;
			END_IF

			IF diBoxLiftFilter.Q AND NOT diLiftBottomFilter.Q  THEN //Error Extra Box on Lift Conveyor
				ErrorID := 7;  //Error Extra Box on Lift Conveyor
				State 	:= ERROR;
			END_IF

			IF diLiftBottom THEN  // Sensor at the Bottom pos
				doConvBottom  	:= TRUE;  // Run the Bottom Conv
				doConvLift     	:= TRUE; //Run the uload Con
			END_IF
			BoxIsPassed := diBoxLiftTON.Q;

			IF diLiftBottom AND ( diBoxLift OR diBoxLiftTON.Q)  AND NOT CounterJamInfeed.Q THEN  // Sensor at the outfeed of the unload conveyor detected
				doConvBottom  	 := FALSE; 	// Stop the Lift Conv
				doLiftBottom	 := FALSE;  //Move the lift conv to unload
				doConvLift       := BoxIsPassed; 	//Stop the uload Con
				State := MAKE;   // Change the state to UnLoad
			END_IF
			IF gUserReset THEN   // RESET Procedure
				gUserReset 	:= FALSE;
				State 		:= STOP;
			END_IF
		UPPER:  //**************** UPPER *********************************************** UPPER ********************************************************************* UPPER

			doLiftTop     := TRUE; //Move the lift conv to Bottom pos

			doConvBottom := NOT diConvBottom; // Stop the bottom conv
			CounterJamInfeed.RESET 	:= FALSE;
			CounterJamInfeed.CU 	:= diConvTopFilter.Q; // Count jammed box
			CounterJamInfeed();
			IF CounterJamInfeed.Q THEN //Infeed Jam Lower code
			     ErrorID 	:= 2;  //Infeed Jam Lower Error
		 	     State 		:= ERROR;
			END_IF
			TimerUpperSensorBlock.IN :=diConvTop AND doConvTop;  // Detect sensor block if the conv run
			TimerUpperSensorBlock();
			IF TimerUpperSensorBlock.Q THEN //Infeed Jam Lower code
				ErrorID 	:= 4;  //Infeed Jam Lower Error
				State 		:= ERROR;
			END_IF
			IF diBoxLiftFilter.Q AND NOT diLiftTopFilter.Q  THEN //Error Extra Box on Lift Conveyor
				ErrorID := 7;  //Error Extra Box on Lift Conveyor
				State 	:= ERROR;
			END_IF

			IF diLiftTop THEN  // Sensor at the Bottom pos
				doConvTop  	 := TRUE;  // Run the Bottom Conv
				doConvLift   := TRUE; //Run the uload Con
			END_IF
			BoxIsPassed := diBoxLiftTON.Q;
			IF diLiftTop AND ( diBoxLift OR diBoxLiftTON.Q) AND NOT CounterJamInfeed.Q THEN  // Sensor at the outfeed of the unload conveyor detected
				doConvTop  	 := FALSE; 	// Stop the Lift Conv
				doLiftTop	 := FALSE;  //Move the lift conv to unload
				doConvLift   := BoxIsPassed; //Stop the uload Con
				State := MAKE;   		// Change the state to UnLoad
			END_IF
			IF gUserReset THEN   // RESET Procedure
				gUserReset 	:= FALSE;
				State 		:= STOP;
			END_IF
		UNLOAD:  //**************** UNLOAD *********************************************** UNLOAD ********************************************************************* UNLOAD

			gActivateMotion := TRUE;
			doLiftUnload	 := TRUE;  //Move the lift conv to unload
			aoConvLiftVelocity		:= UserConvLiftVelocity +  ( gMpAxisBasic_Axis1.Velocity / 1000.0 * gSpeedFactor);

			CounterJamInfeed.RESET 	:= FALSE;
			CounterJamInfeed.CU 	:= EDGENEG(diBoxLiftFilter.Q); // Extra box on conv lift
			CounterJamInfeed();
			IF CounterJamInfeed.Q THEN
				ErrorID := 7;  //Extra box on conv lift
				State 	:= ERROR;
			END_IF

			doConvTop    := NOT diConvTop ;   // Stop the Top Conv
			doConvBottom := NOT diConvBottom; // Stop the bottom conv

			IF ( diLiftUnload OR Test_Bit_0) THEN  // Sensor at the center of the unload conveyor detected
				doConvLift  	 := TRUE;  // Run the Lift Conv
			END_IF

			IF diUnloaded AND diLiftUnload THEN  // Sensor at the outfeed of the unload conveyor detected
				doConvLift  	 := FALSE; // Stop the Lift Conv
				doLiftUnload	 := FALSE;  //Move the lift conv to unload
				gActivateMotion := FALSE;
				State := MAKE;   // Change the state to UnLoad
			END_IF

			IF gUserReset THEN   // RESET Procedure
				gUserReset := FALSE;
				State := STOP;
			END_IF

		ERROR: //**************** ERROR *********************************************** ERROR ********************************************************************* ERROR
			aoConvTopVelocity 			:= 0.0;   	// Turn off the Conv Top
			aoInfeedConvTopVelocity  	:= 0.0; 	// Turn off the Infeed Conv Top
			aoConvLiftVelocity 			:= 0.0; 	// Turn off the Conv Lift
			aoInfeedConvBottomVelocity 	:= 0.0; 	// Turn off the Infeed Conv Bottom
			aoOutfeedConvVelocity 		:= 0.0; 	// Turn off outfeed Conv
			aoConvBottomVelocity  		:= 0.0;  	 // Turn off the Conv Top
			doLiftUnload 				:= FALSE; 	 //Lift Unload Position Cmd
			doLiftTop 					:= FALSE; 	//Lift Top Position Cmd
			doLiftBottom 				:= FALSE; //Lift Bottom Position Cmd
			doConvTop 					:= FALSE; //Top Conveyor Run Cmd
			doConvLift 					:= FALSE; //Lift Conveyor Run Cmd
			doConvBottom 				:= FALSE; //Bottom Conveyor Run
			//Alarm Image
			gDispalyAlarm 				:= gDisplayBlink;	//Dispaly Alarm Image
			gDispalyStop 				:= TRUE; 	// Dispaly Stop Image
			gDispalyRun 				:= FALSE;   // Not Dispaly Run Image
			SaveAlarm 					:= TRUE;

			IF i<>0 THEN
				gErrorTime[i] 		:= gErrorTime[i-1];  // Shift Error Time
				gErrorDes[i] 		:= gErrorDes[i-1];    // Shift Error Description
				ErrorTimeString[i] := ErrorTimeString[i-1]; //To dispaly in mappView
				i := i-1;
			END_IF
			IF i=0 THEN
				CopyDone := TRUE;
			END_IF
			IF SaveAlarm AND EDGEPOS(CopyDone) THEN
				gErrorDes[0] 		:= ErrorTable[ErrorID]; // Save Current Error
				DTGetTime_0.enable 	:= TRUE;
				DTGetTime_0();
				gErrorTime[0]:=DTGetTime_0.DT1;  // Save Current Time
				ErrorTimeString[0] 	:= DT_TO_STRING(gErrorTime[0]); //To dispaly in mappView
			END_IF

			IF gUserReset THEN   // RESET Procedure
				gUserReset 			:= FALSE; // Reset Request disable
				DTGetTime_0.enable	:=FALSE; // Function save time Request disable
				SaveAlarm 			:= FALSE;  // Saving Finish
				CopyDone 			:= FALSE;  //Copy previous alarm Done
				ErrorID 			:= 0;  //Infeed Jam Lower Error
				gDispalyNoComm 		:= FALSE; // Disaply off for communication error
				State 				:= STOP;
				i:=9;
			END_IF

		INIT:

			IF  gServoInitialized THEN
				State := STOP;
			END_IF

	END_CASE //*********************************************************************** END CASE

	/// Recepit Management ********************************************************Recepit Management**************************************************************************************

	IF  gReceiptChanged THEN
		 UserConvTopVelocity       	    := gSiPhysics[gSpeedRefHmi].UserConvTopVelocity   ;   // Load Speed the Conv Top
		 UserConvBottomVelocity		    := gSiPhysics[gSpeedRefHmi].UserConvBottomVelocity;   // Load Speed the Conv Top
		 UserConvLiftVelocity			:= gSiPhysics[gSpeedRefHmi].UserConvLiftVelocity ; // Load Speed the Conv Lift
		 UserOutfeedConvVelocity 		:= gSiPhysics[gSpeedRefHmi].UserOutfeedConvVelocity; // Load Speed outfeed Conv
		 UserInfeedConvTopVelocity 		:= gSiPhysics[gSpeedRefHmi].UserInfeedConvTopVelocity; // Load Speed the Infeed Conv Top
		 UserInfeedConvBottomVelocity 	:= gSiPhysics[gSpeedRefHmi].UserInfeedConvBottomVelocity; // Load Speed the Infeed Conv Bottom
		 UserTopBoxReleaseTime 			:= gSiPhysics[gSpeedRefHmi].UserTopBoxReleaseTime;  //Load Release Speed
	     UserBottomBoxReleaseTime 		:= gSiPhysics[gSpeedRefHmi].UserBottomBoxReleaseTime; //Load Release Speed
		 gReceiptChanged := FALSE;
	END_IF

	IF gSaveParameter THEN
		gSiPhysics[gSpeedRefHmi].UserConvTopVelocity       	    := UserConvTopVelocity   ;   // Set Speed the Conv Top
		gSiPhysics[gSpeedRefHmi].UserConvBottomVelocity		    := UserConvBottomVelocity;   // Set Speed the Conv Top
		gSiPhysics[gSpeedRefHmi].UserConvLiftVelocity			:= UserConvLiftVelocity ; // Set Speed the Conv Lift
		gSiPhysics[gSpeedRefHmi].UserOutfeedConvVelocity 		:= UserOutfeedConvVelocity; // Set Speed outfeed Conv
		gSiPhysics[gSpeedRefHmi].UserInfeedConvTopVelocity 		:= UserInfeedConvTopVelocity; // Set Speed the Infeed Conv Top
		gSiPhysics[gSpeedRefHmi].UserInfeedConvBottomVelocity 	:= UserInfeedConvBottomVelocity; // Set Speed the Infeed Conv Bottom
		gSiPhysics[gSpeedRefHmi].UserTopBoxReleaseTime 			:= UserTopBoxReleaseTime;  //Box Release Speed
		gSiPhysics[gSpeedRefHmi].UserBottomBoxReleaseTime 		:= UserBottomBoxReleaseTime; //Box Release Speed
		gSaveParameter := FALSE;
	END_IF

	SpeedInfoText := SpeedInfoTextTable[gSpeedRefHmi];  // Dispaly speed info

	// Information Dispaly **********************************************Information Dispaly************************************************************************************************
	gBoxCountUnload.CU 		:= diUnloaded;  // Count Unloaded Box
	gBoxCountUnload.RESET 	:= ResetCount; // Reset from Dispaly
	gBoxCountUnload();
	BoxCountUnloadDis 		:= gBoxCountUnload.CV ; // Dispaly Count

	StatusDispaly 			:= StatusDispalyDefault[State];  // Dispaly Status on the main page
	StatusDispalyTopContent := StatusDispalyTopContentDefault[State];// Dispaly Status on the top page

	// Find Box per minutes
	oneMinTimer.IN := TRUE;
	oneMinTimer();
	IF EDGEPOS(oneMinTimer.Q) THEN
		oneMinTimer.IN := FALSE;
		oneMinTimer();
		TotalBoxUnloaded := gBoxCountUnload.CV - PrevBoxCountUnload;  // how maney box uloaded last 10s
		PrevBoxCountUnload :=gBoxCountUnload.CV;
		Performance := TotalBoxUnloaded*6; // how maney box uloaded last 60s
		IF Performance > gSiPhysics[gSpeedRefHmi].MaximumUloadedBox THEN  // Save only if the new value is greater than the previous to keep the maximum
			gSiPhysics[gSpeedRefHmi].MaximumUloadedBox := Performance;
		END_IF
	END_IF
	// Dispaly XY Chart
	DispalyGraph[0]:= 1;  // for X0 chart
	DispalyGraph[1]:= 2;  // for X1 chart
	DispalyGraph[2]:= 3;  // for X2 chart
	TotalBoxUnloadedPerSpeed[0] := gSiPhysics[0].MaximumUloadedBox  ;  // how maney box uloaded last 10s per Low speed
	TotalBoxUnloadedPerSpeed[1] := gSiPhysics[1].MaximumUloadedBox  ;  // how maney box uloaded last 10s per Medium speed
	TotalBoxUnloadedPerSpeed[2] := gSiPhysics[2].MaximumUloadedBox  ;  // how maney box uloaded last 10s per High speed
	// Dispaly Bar Chart
	TotalBoxUnloadedPerSpeedLow  	 := gSiPhysics[0].MaximumUloadedBox;  // how maney box uloaded last 10s per Low speed
	TotalBoxUnloadedPerSpeedMeduim	 := gSiPhysics[1].MaximumUloadedBox;  // how maney box uloaded last 10s per Medium speed
	TotalBoxUnloadedPerSpeedHigh	 := gSiPhysics[2].MaximumUloadedBox;  // how maney box uloaded last 10s per High speed

	// di Sensors noise filter

	diBoxLiftFilter.IN := diBoxLift;    //di Sensors noise filter
	diBoxLiftFilter();

	diLiftTopFilter.IN := diLiftTop; //di Sensors noise filter
	diLiftTopFilter();

	diLiftBottomFilter.IN := diLiftBottom; //di Sensors noise filter
	diLiftBottomFilter();

	diConvBottomFilter.IN := diConvBottom; //di Sensors noise filter
	diConvBottomFilter();

	diConvTopFilter.IN := diConvTop; //di Sensors noise filter
	diConvTopFilter();

	// if doConvTop doConvLift then we can assume the box is in the begging of the conv lift
	diBoxLiftTON.IN := ((doConvLift AND doConvTop AND State = UPPER ) OR (doConvLift AND doConvBottom AND State = LOWER))  ;
	diBoxLiftTON();

END_PROGRAM
```

#### Exit.st
```iecst
PROGRAM _EXIT
	(* Insert code here *)
	 //
	aoConvTopVelocity 			:= 0.0;   	// Turn off the Conv Top
	aoInfeedConvTopVelocity  	:= 0.0; 	// Turn off the Infeed Conv Top
	aoConvLiftVelocity 			:= 0.0; 	// Turn off the Conv Lift
	aoInfeedConvBottomVelocity 	:= 0.0; 	// Turn off the Infeed Conv Bottom
	aoOutfeedConvVelocity 		:= 0.0; 	// Turn off outfeed Conv
	aoConvBottomVelocity  		:= 0.0;  	 // Turn off the Conv Top
	doLiftUnload 				:= FALSE; 	 //Lift Unload Position Cmd
	doLiftTop 					:= FALSE; 	//Lift Top Position Cmd
	doLiftBottom 				:= FALSE; //Lift Bottom Position Cmd
	doConvTop 					:= FALSE; //Top Conveyor Run Cmd
	doConvLift 					:= FALSE; //Lift Conveyor Run Cmd
	doConvBottom 				:= FALSE; //Bottom Conveyor Run

END_PROGRAM
```

#### Init.st
```iecst
PROGRAM _INIT
	(* Insert code here *)

	// load parameter first time
	UserConvTopVelocity       	    := gSiPhysics[gSpeedRefHmi].UserConvTopVelocity   ;   // Load Speed the Conv Top
	UserConvBottomVelocity		    := gSiPhysics[gSpeedRefHmi].UserConvBottomVelocity;   // Load Speed the Conv Top
	UserConvLiftVelocity			:= gSiPhysics[gSpeedRefHmi].UserConvLiftVelocity ; // Load Speed the Conv Lift
	UserOutfeedConvVelocity 		:= gSiPhysics[gSpeedRefHmi].UserOutfeedConvVelocity; // Load Speed outfeed Conv
	UserInfeedConvTopVelocity 		:= gSiPhysics[gSpeedRefHmi].UserInfeedConvTopVelocity; // Load Speed the Infeed Conv Top
	UserInfeedConvBottomVelocity 	:= gSiPhysics[gSpeedRefHmi].UserInfeedConvBottomVelocity; // Load Speed the Infeed Conv Bottom
	UserTopBoxReleaseTime 			:= gSiPhysics[gSpeedRefHmi].UserTopBoxReleaseTime;  //Load Release Speed
	UserBottomBoxReleaseTime 		:= gSiPhysics[gSpeedRefHmi].UserBottomBoxReleaseTime; //Load Release Speed
	gReceiptChanged					:= FALSE;
	aoConvTopVelocity 				:= 0.0;   // Turn off the Conv Top
	aoInfeedConvTopVelocity 		:= 0.0; // Turn off the Infeed Conv Top
	aoConvLiftVelocity 				:= 0.0; // Turn off the Conv Lift
	aoInfeedConvBottomVelocity 		:= 0.0; // Turn off the Infeed Conv Bottom
	aoOutfeedConvVelocity 			:= 0.0; // Turn off outfeed Conv
	aoConvBottomVelocity  			:= 0.0;   // Turn off the Conv Top
	doLiftUnload 					:= FALSE;  //Lift Unload Position Cmd
	doLiftTop 						:= FALSE; //Lift Top Position Cmd
	doLiftBottom 					:= FALSE; //Lift Bottom Position Cmd
	doConvTop 						:= FALSE; //Top Conveyor Run Cmd
	doConvLift 						:= FALSE; //Lift Conveyor Run Cmd
	doConvBottom 					:= FALSE; //Bottom Conveyor Run
	/// STOP Animation
	gDispalyStop 					:= TRUE; 	// Dispaly Stop Image
	gDispalyRun 					:= FALSE;   // Not Dispaly Run Image
	gDispalyAlarm 					:=FALSE;  // Not Dispaly Alarm Image
	gUserStop 						:= FALSE;

END_PROGRAM
```

### Program Logical/AlarmBlink (IEC) - Alarm Pulse

#### Variables.var
```iecst
VAR
	TON_DelayDo1 : TON;
	DelayBlink : TIME := T#500ms;
END_VAR
```

#### Cyclic.st
```iecst
PROGRAM _CYCLIC
	(* Insert code here *)
	TON_DelayDo1.PT := DelayBlink;
// Create Pulse Generator Start

	IF TON_DelayDo1.ET <> DelayBlink THEN
		TON_DelayDo1.IN := TRUE;
	END_IF

	TON_DelayDo1();

	IF EDGEPOS(TON_DelayDo1.Q) THEN
		gDisplayBlink := NOT gDisplayBlink;
		TON_DelayDo1.IN := FALSE;
	END_IF

// Create Pulse Generator End

END_PROGRAM
```

### Program Logical/RecipeMgmt (IEC) - Manage Recipe

#### Variables.var
```iecst
VAR
	State : State_enum;
	uiLoad : BOOL;
	uiSave : BOOL;
	sDeviceName : STRING[255] := 'SIM_Recipes';
	sFileName : STRING[255] := 'recipe1';
	sVariableName : STRING[255] := 'gSiPhysics';
	MpRecipeCsv_0 : MpRecipeCsv;
	MpRecipeRegPar_0 : MpRecipeRegPar;

	RecipeError : BOOL;
	ErrorReset : BOOL;
END_VAR
```

#### Cyclic.ld
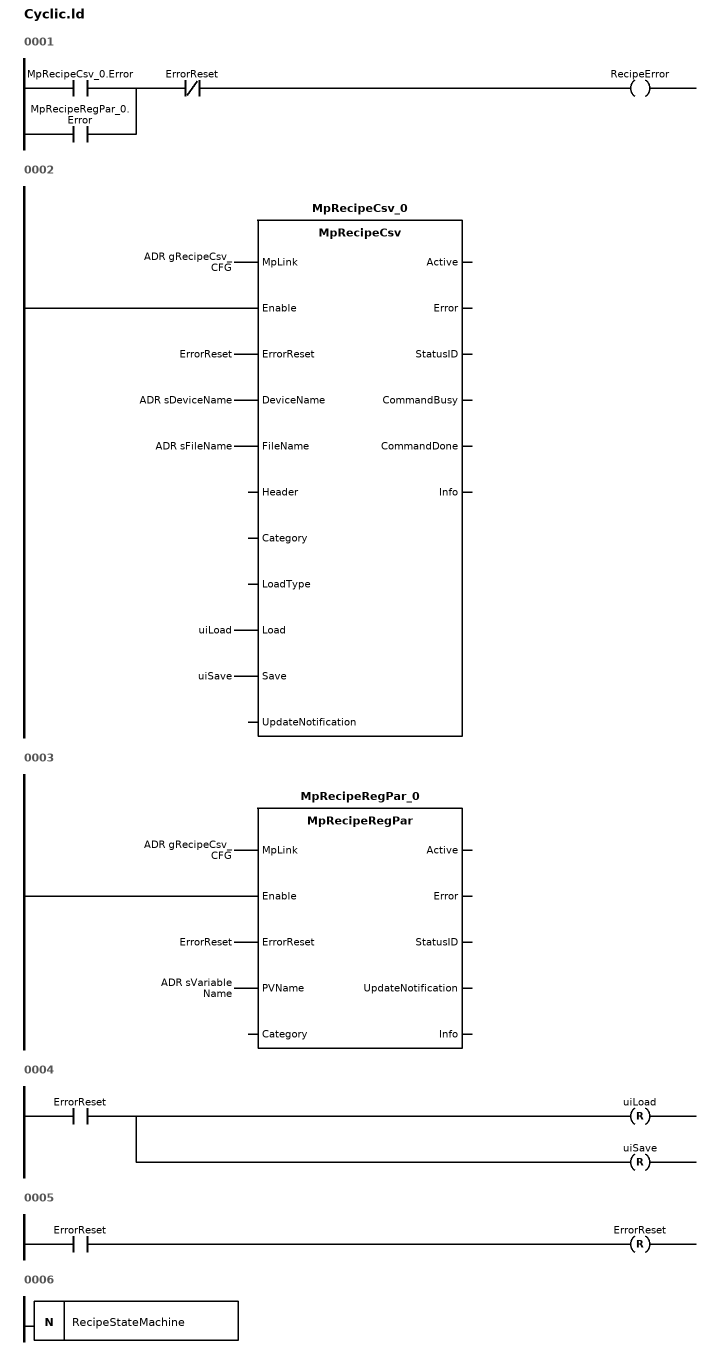
Ladder, written as Structured Text:
```iecst
PROGRAM _CYCLIC
(* Network 1 *)
RecipeError := (MpRecipeCsv_0.Error OR MpRecipeRegPar_0.Error) AND NOT ErrorReset;

(* Network 2 *)
MpRecipeCsv_0(MpLink := ADR(gRecipeCsv_CFG), Enable := TRUE, ErrorReset := ErrorReset, DeviceName := ADR(sDeviceName), FileName := ADR(sFileName), Load := uiLoad, Save := uiSave);

(* Network 3 *)
MpRecipeRegPar_0(MpLink := ADR(gRecipeCsv_CFG), Enable := TRUE, ErrorReset := ErrorReset, PVName := ADR(sVariableName));

(* Network 4 *)
IF ErrorReset THEN
    uiLoad := FALSE;
    uiSave := FALSE;
END_IF;

(* Network 5 *)
IF ErrorReset THEN ErrorReset := FALSE; END_IF;

(* Network 6 *)
RecipeStateMachine;
END_PROGRAM
```

#### RecipeStateMachine.st
```iecst
ACTION RecipeStateMachine:

	CASE State OF
	//**************************************************LOAD**************
		LOAD:
			IF MpRecipeCsv_0.CommandDone THEN
				State := WAIT;
				uiLoad := FALSE;
			END_IF
	//**************************************************SAVE***************
		SAVE:
			IF MpRecipeCsv_0.CommandDone THEN
				State := WAIT;
				uiSave := FALSE;
			END_IF

	//**************************************************WAIT***************
		WAIT:
			IF (NOT MpRecipeCsv_0.CommandBusy AND uiLoad) THEN
				State := LOAD;
			END_IF
			IF (NOT MpRecipeCsv_0.CommandBusy AND uiSave) THEN
				State := SAVE;
			END_IF

	END_CASE

END_ACTION
```

### Data object Logical/Cam (Cam) - Cam - Lift Speed

#### Cam.cam
```
CamProfile (NcSwId=ACP10, MasterAxisVelocity=1, MasterAxisAcceleration=0, DefaultCurveType=Polynomial5, MathematicalNotation=true)
  FixPoint (x=0, IsMathX=true, y=0, IsDefinedDy=true, Dy=0, IsMathDy=true, IsDefinedDdy=false, Ddy=0, IsMathDdy=true, IsDefinedDddy=false, Dddy=0, IsMathDddy=true)
  FixPoint (x=1, IsMathX=true, y=1, IsDefinedDy=false, Dy=0, IsMathDy=true, IsDefinedDdy=false, Ddy=0, IsMathDdy=true, IsDefinedDddy=false, Dddy=0, IsMathDddy=true)
  Curve (Type=Polynomial5)
    LeftBoundary (IsDefinedDdy=false, Ddy=0, IsMathDdy=true, IsDefinedDddy=false, Dddy=0, IsMathDddy=true)
    RightBoundary (IsDefinedDdy=false, Ddy=0, IsMathDdy=true, IsDefinedDddy=false, Dddy=0, IsMathDddy=true)
    Spline3 (IsContinuous4Derivative=false, IsDefinedSaddlePoint=false, IsDefinedLineAs2ndSegment=false, IsDefinedSlopeOfLine=false, SlopeOfLine=0, IsMathSlopeOfLine=true)
    Supremum (y=1.7e+308, Dy=1.7e+308, IsMathDy=true, Ddy=1.7e+308, IsMathDdy=true, Dddy=1.7e+308, IsMathDddy=true)
    Infimum (y=-1.7e+308, Dy=-1.7e+308, IsMathDy=true, Ddy=-1.7e+308, IsMathDdy=true, Dddy=-1.7e+308, IsMathDddy=true)
  Cam (LeftBoundaryIndex=0, RightBoundaryIndex=1)
    Supremum (y=1.7e+308, Dy=1.7e+308, IsMathDy=true, Ddy=1.7e+308, IsMathDdy=true, Dddy=1.7e+308, IsMathDddy=true)
    Infimum (y=-1.7e+308, Dy=-1.7e+308, IsMathDy=true, Ddy=-1.7e+308, IsMathDdy=true, Dddy=1.7e+308, IsMathDddy=true)
  ChartExtensions
```

### Program Logical/Axis1ST (IEC) - Ctrl of the Axis 1

#### Variables.var
```iecst
VAR CONSTANT
	STATE_HOME : USINT := 2;
	STATE_POWER_ON : USINT := 1;
	STATE_ERROR : USINT := 101;
	STATE_JOG : USINT := 17;
	STATE_MOVE_ABSOLUTE : USINT := 14;
	STATE_STOP : USINT := 11;
	STATE_WAIT : USINT := 0;
	STATE_READY : USINT := 10;
END_VAR
VAR
	AxisStep : UINT;
	Axis1_ErrorID : UINT;
	Axis2Home : BOOL;
	Axis1Home : BOOL;
	Test_bit_2 : BOOL;
END_VAR
```

#### Cyclic.st
```iecst
PROGRAM _CYCLIC
	(* Insert code here *)

	gMpAxisBasic_Axis1.MpLink 			:= ADR(gAxis1_MpLink);
	gMpAxisBasic_Axis1.Enable 			:= TRUE;
	gMpAxisBasic_Axis1.Parameters 		:= ADR(gMpAxisBasicParType_Axis1);

	gMpAxisBasic_AxisVirtu.MpLink 		:= ADR(gAxisV_MpLink);
	gMpAxisBasic_AxisVirtu.Enable 		:= TRUE;
	gMpAxisBasic_AxisVirtu.Parameters 	:= ADR(gMpAxisBasicParType_AxisVirtu);

	gMpAxisCoupling_0.MpLink 			:= ADR(gAxis1_MpLink);
	gMpAxisCoupling_0.MpLinkMaster 		:= ADR(gAxisV_MpLink);

	gCouplingPar.Cam.ID					:= 1;
	gMpAxisCoupling_0.Parameters		:= ADR(gCouplingPar);

	CASE AxisStep OF

		STATE_WAIT :     //**************** 00000 ************************** STATE_WAIT ********************* 0000 ********************* STATE_WAIT
			gMpAxisBasic_Axis1.Power		:= FALSE;
			gMpAxisBasic_AxisVirtu.Power	:= FALSE;
			gMpAxisCoupling_0.Enable 	:= FALSE;
			IF (Axis1.Exists AND NOT gMpAxisCoupling_0.Active AND gServoInitialized) THEN
				AxisStep :=  STATE_POWER_ON;
			END_IF

		STATE_POWER_ON : //************************ 1 ****************** STATE_POWER_ON ********************* 1 ********************* STATE_POWER_ON
				gMpAxisBasic_Axis1.Power		:= TRUE;
				gMpAxisBasic_AxisVirtu.Power	:= TRUE;
			IF (gMpAxisBasic_Axis1.PowerOn = TRUE AND gMpAxisBasic_AxisVirtu.PowerOn = TRUE  ) THEN
					Axis1Home		:= FALSE;
					Axis2Home		:= FALSE;
					AxisStep := STATE_HOME;

     		END_IF

			IF (gMpAxisBasic_Axis1.Error OR gMpAxisBasic_Axis2.Error) THEN
				Axis1_ErrorID := 1;
				AxisStep := STATE_ERROR;
			END_IF

		STATE_HOME :  //***************************** 2 ********************STATE_HOME************************* 2 *********************STATE_HOME

			Axis1.statusHomed 				:= FALSE;
			IF NOT gMpAxisCoupling_0.Active THEN
			gMpAxisBasic_Axis1.Home 		:= TRUE;
				gMpAxisBasicParType_Axis1.Homing.Mode 		:= mcHOMING_DIRECT;
				gMpAxisBasicParType_Axis1.Homing.Position 	:= 0.0;
				gMpAxisBasic_AxisVirtu.Home 		:= TRUE;
				gMpAxisBasicParType_AxisVirtu.Homing.Mode 		:= mcHOMING_DIRECT;
				gMpAxisBasicParType_AxisVirtu.Homing.Position 	:= 0.0;
			END_IF

			IF EDGEPOS(gMpAxisBasic_Axis1.IsHomed) THEN
				Axis1Home		:= TRUE;
			END_IF
			IF EDGEPOS(gMpAxisBasic_AxisVirtu.IsHomed) THEN
				Axis2Home		:= TRUE;
			END_IF

			IF (Axis1Home AND Axis2Home   ) THEN
				Axis1.statusHomed 			:= 1;
				gMpAxisBasic_Axis1.Home 	:= FALSE;
				gMpAxisBasic_AxisVirtu.Home := FALSE;
				gMpAxisCoupling_0.Enable 	:= TRUE;
				AxisStep := STATE_READY;
			END_IF

			IF (gMpAxisBasic_Axis1.Error) THEN
				Axis1_ErrorID := 2;
				AxisStep := STATE_ERROR;
			END_IF

		STATE_READY : //***************************** 10 ************************ STATE_READY ******************** 10 ************************** STATE_READY

			Axis1.statusStarting :=0;
			IF (Axis1.cmdHome = 1 )THEN
				Axis1Home					:= FALSE;
				Axis2Home					:= FALSE;
				Axis1.cmdHome		 		:= FALSE;
				gMpAxisCoupling_0.Enable	:= FALSE;
				gMpAxisCoupling_0.Cam 		:= FALSE;
				AxisStep 				:= STATE_HOME;
			ELSIF (Axis1.cmdStop = 1) THEN
				gMpAxisCoupling_0.Cam 		:= FALSE;
				AxisStep 				:= STATE_WAIT;
				Axis1.cmdStop 			:= FALSE;
			ELSIF (Axis1.cmdManualForward  AND gMpAxisCoupling_0.Active) THEN
				gMpAxisCoupling_0.Cam 	:=TRUE;
				AxisStep := STATE_JOG;
			END_IF

			IF gMpAxisBasic_Axis1.Error THEN
				AxisStep := STATE_ERROR;
			END_IF

		STATE_STOP : //*********************** 11 ****************************** STATE_STOP ***************************** 11 ********************** STATE_STOP

			gMpAxisBasic_AxisVirtu.Stop := TRUE;
			(* if axis is stopped go to state wait *)
			IF (gMpAxisBasic_AxisVirtu.Stopped = 1  ) THEN
				gMpAxisBasic_AxisVirtu.Stop := 0;
				AxisStep := STATE_READY;
			END_IF
			(* check if error occured *)
			IF (gMpAxisBasic_Axis1.Error ) THEN
				Axis1_ErrorID := 3;
				AxisStep := STATE_ERROR;
			END_IF

		STATE_JOG : //************************* 17 **************************** STATE_JOG ********************************* 17 ********************* STATE_JOG

			IF ( Axis1.cmdManualForward  AND gMpAxisCoupling_0.InSync) THEN
				gMpAxisBasic_AxisVirtu.MoveAdditive:= TRUE;
			END_IF

			IF NOT(Axis1.cmdManualForward ) THEN
				gMpAxisBasic_AxisVirtu.MoveAdditive:= FALSE;
//				Axis1Home					:= FALSE;
//				Axis2Home					:= FALSE;
//				Axis1.cmdHome		 		:= FALSE;
				IF (NOT gMpAxisBasic_AxisVirtu.CommandBusy AND NOT gMpAxisBasic_Axis1.CommandBusy) THEN
					AxisStep 				:= STATE_READY;
//					gMpAxisCoupling_0.Enable	:= FALSE;
//					gMpAxisCoupling_0.Cam 		:= FALSE;
				END_IF
//				AxisStep := STATE_READY;
			END_IF

			(* check if error occured *)
			IF (gMpAxisBasic_Axis1.Error OR gMpAxisBasic_Axis2.Error) THEN
				Axis1_ErrorID := 4;
				AxisStep := STATE_ERROR;
			END_IF

		STATE_ERROR : //********************** 101 ******************************* STATE_ERROR **************************** 101 ********************** STATE_ERROR

			Axis1.statusStarting 		:=0;
			Axis1.statusFaulted 		:= TRUE;
			gMpAxisCoupling_0.Gear 		:= FALSE;
			gMpAxisCoupling_0.Cam 		:= FALSE;
			gMpAxisBasic_Axis1.Power 	:= FALSE;
			gMpAxisBasic_Axis1.Home 	:= FALSE;
			gMpAxisBasic_Axis1.Stop 	:= FALSE;
			gMpAxisBasic_AxisVirtu.Power 		:= FALSE;
			gMpAxisBasic_AxisVirtu.Home 		:= FALSE;
			gMpAxisBasic_AxisVirtu.Stop 		:= FALSE;
			gMpAxisBasic_Axis1.MoveAbsolute 	:= FALSE;
			gMpAxisBasic_AxisVirtu.MoveVelocity := FALSE;
			gMpAxisBasic_AxisVirtu.MoveAbsolute := FALSE;
			gMpAxisBasic_AxisVirtu.MoveVelocity := FALSE;
			gMpAxisBasic_Axis1.ErrorReset 		:= TRUE;
			gMpAxisBasic_AxisVirtu.ErrorReset 	:= TRUE;
			gMpAxisCoupling_0.ErrorReset   		:= TRUE;

			IF (NOT(gMpAxisBasic_Axis1.Error ) AND NOT(gMpAxisBasic_AxisVirtu.Error )) THEN
				Axis1.statusFaulted:=FALSE;
				gMpAxisBasic_Axis1.ErrorReset 		:= FALSE;
				gMpAxisBasic_AxisVirtu.ErrorReset 	:= FALSE;
				gMpAxisCoupling_0.ErrorReset   		:= FALSE;
				AxisStep := STATE_WAIT;
				Axis1.statusErrorID := 0;
			END_IF

	END_CASE

	gMpAxisBasic_Axis1();
	gMpAxisBasic_Axis2();
	gMpAxisBasic_AxisVirtu();
	gMpAxisCoupling_0();

	Axis1.cmdManualForward 	:= gActivateMotion;

END_PROGRAM
```

#### Exit.st
```iecst
PROGRAM _EXIT
	(* Insert code here *)
	gMpAxisBasic_Axis1.Enable 		:= FALSE;
	gMpAxisBasic_Axis1();
	gMpAxisBasic_AxisVirtu.Enable 		:= TRUE;
	gMpAxisBasic_AxisVirtu();
	gMpAxisCoupling_0.Enable			:= FALSE;
	gMpAxisCoupling_0();
END_PROGRAM
```

#### Init.st
```iecst
PROGRAM _INIT
	(* Insert code here *)
	gMpAxisBasicParType_Axis2.AutoTune.Mode 				:= mcAXIS_TUNE_AUTOMATIC;
	gMpAxisBasicParType_Axis2.AutoTune.MaxCurrentPercent 	:= 80.0;
	gMpAxisBasicParType_Axis2.AutoTune.MaxDistance 			:= 10;
	gMpAxisBasicParType_Axis2.AutoTune.MaxPositionError 	:= 30;

	gMpAxisBasicParType_Axis1.AutoTune.Mode 				:= mcAXIS_TUNE_AUTOMATIC;
	gMpAxisBasicParType_Axis1.AutoTune.MaxCurrentPercent 	:= 80.0;
	gMpAxisBasicParType_Axis1.AutoTune.MaxDistance 			:= 10;
	gMpAxisBasicParType_Axis1.AutoTune.MaxPositionError 	:= 30;

	Axis1.Exists := TRUE;
	gMpAxisBasicParType_AxisVirtu.Position := 360.0;
	gMpAxisBasicParType_AxisVirtu.Distance := 360.0;
	gMpAxisBasicParType_AxisVirtu.Velocity := 360.0;
	gMpAxisBasicParType_AxisVirtu.Deceleration := 1500;
	gMpAxisBasicParType_AxisVirtu.Acceleration := 1500;
	gCouplingPar.Cam.MasterScaling := 36000;
	gCouplingPar.Cam.SlaveScaling := 36000;

END_PROGRAM
```

### Program Logical/PowerON (IEC) - PowerOnTimer

#### Variables.var
```iecst
VAR
	ObjectPassed : BOOL;
	TON_DelayDo1 : TON;
	CTU_CountDO1 : CTU;
	DelayOpc : TIME := T#20s;
	StartTimer : BOOL;
	DelayPulse : BOOL;
	ErrorAxis12 : LREAL;
END_VAR
```

#### Cyclic.st
```iecst
PROGRAM _CYCLIC
	(* Insert code here *)
	TON_DelayDo1.PT := DelayOpc;
// Create Pulse Generator Start

	IF TON_DelayDo1.ET <> DelayOpc THEN
		TON_DelayDo1.IN := TRUE;
	END_IF

	TON_DelayDo1();
	gServoInitialized:= TON_DelayDo1.Q ;

// Create Pulse Generator End

END_PROGRAM
```

#### Init.st
```iecst
PROGRAM _INIT
	(* Insert code here *)

END_PROGRAM
```

### Program Logical/CamAutomat (IEC) - Test with Cam automat

#### Variables.var
```iecst
VAR CONSTANT
	STATE_HOME : USINT := 2;
	STATE_POWER_ON : USINT := 1;
	STATE_ERROR : USINT := 101;
	STATE_JOG : USINT := 17;
	STATE_MOVE_ABSOLUTE : USINT := 14;
	STATE_STOP : USINT := 11;
	STATE_WAIT : USINT := 0;
	STATE_READY : USINT := 10;
END_VAR
VAR
	AxisStep : UINT;
	Axis3_ErrorID : UINT;
	Axis2Home : BOOL;
	Axis1Home : BOOL;
	Test_bit_2 : BOOL;
END_VAR
```

#### Cyclic.st
```iecst
PROGRAM _CYCLIC
	(* Insert code here *)

	gMpAxisBasic_Axis3.MpLink 			:= ADR(gAxis3_MpLink);
	gMpAxisBasic_Axis3.Enable 			:= TRUE;
	gMpAxisBasic_Axis3.Parameters 		:= ADR(gMpAxisBasicParType_Axis3);

	gMpAxisBasic_AxisVirtu3.MpLink 		:= ADR(gAxisV3_MpLink);
	gMpAxisBasic_AxisVirtu3.Enable 		:= TRUE;
	gMpAxisBasic_AxisVirtu3.Parameters 	:= ADR(gMpAxisBasicParType_AxisVirtu3);

	gMpAxisCoupling_3.MpLink 			:= ADR(gAxis3_MpLink);
	gMpAxisCoupling_3.MpLinkMaster 		:= ADR(gAxisV3_MpLink);

	gCouplingPar3.Cam.ID				:= 1;
	gMpAxisCoupling_3.Parameters		:= ADR(gCouplingPar3);

	CASE AxisStep OF

		STATE_WAIT :     //**************** 00000 ************************** STATE_WAIT ********************* 0000 ********************* STATE_WAIT
			gMpAxisBasic_Axis3.Power		:= FALSE;
			gMpAxisBasic_AxisVirtu3.Power	:= FALSE;
			gMpAxisCoupling_3.Enable 	:= FALSE;
			IF (Axis3.Exists AND NOT gMpAxisCoupling_3.Active AND gServoInitialized) THEN
				AxisStep :=  STATE_POWER_ON;
			END_IF

		STATE_POWER_ON : //************************ 1 ****************** STATE_POWER_ON ********************* 1 ********************* STATE_POWER_ON
			gMpAxisBasic_Axis3.Power		:= TRUE;
			gMpAxisBasic_AxisVirtu3.Power	:= TRUE;
			IF (gMpAxisBasic_Axis3.PowerOn = TRUE AND gMpAxisBasic_AxisVirtu3.PowerOn = TRUE  ) THEN
				Axis1Home		:= FALSE;
				Axis2Home		:= FALSE;
				AxisStep := STATE_HOME;

			END_IF

			IF (gMpAxisBasic_Axis3.Error OR gMpAxisBasic_Axis3.Error) THEN
				Axis3_ErrorID := 1;
				AxisStep := STATE_ERROR;
			END_IF

		STATE_HOME :  //***************************** 2 ********************STATE_HOME************************* 2 *********************STATE_HOME

			Axis3.statusHomed 				:= FALSE;
			IF NOT gMpAxisCoupling_3.Active THEN
				gMpAxisBasic_Axis3.Home 		:= TRUE;
				gMpAxisBasicParType_Axis3.Homing.Mode 		:= mcHOMING_DIRECT;
				gMpAxisBasicParType_Axis3.Homing.Position 	:= 0.0;
				gMpAxisBasic_AxisVirtu3.Home 		:= TRUE;
				gMpAxisBasicParType_AxisVirtu3.Homing.Mode 		:= mcHOMING_DIRECT;
				gMpAxisBasicParType_AxisVirtu3.Homing.Position 	:= 0.0;
			END_IF

			IF EDGEPOS(gMpAxisBasic_Axis3.IsHomed) THEN
				Axis1Home		:= TRUE;
			END_IF
			IF EDGEPOS(gMpAxisBasic_AxisVirtu3.IsHomed) THEN
				Axis2Home		:= TRUE;
			END_IF

			IF (Axis1Home AND Axis2Home   ) THEN
				Axis3.statusHomed 			:= 1;
				gMpAxisBasic_Axis3.Home 	:= FALSE;
				gMpAxisBasic_AxisVirtu3.Home := FALSE;
				gMpAxisCoupling_3.Enable 	:= TRUE;
				AxisStep := STATE_READY;
			END_IF

			IF (gMpAxisBasic_Axis3.Error) THEN
				Axis3_ErrorID := 2;
				AxisStep := STATE_ERROR;
			END_IF

		STATE_READY : //***************************** 10 ************************ STATE_READY ******************** 10 ************************** STATE_READY

			Axis3.statusStarting :=0;
			IF (Axis3.cmdHome = 1 )THEN
				Axis1Home					:= FALSE;
				Axis2Home					:= FALSE;
				Axis3.cmdHome		 		:= FALSE;
				gMpAxisCoupling_3.Enable	:= FALSE;
				gMpAxisCoupling_3.Cam 		:= FALSE;
				AxisStep 				:= STATE_HOME;
			ELSIF (Axis3.cmdStop = 1) THEN
				gMpAxisCoupling_3.Cam 		:= FALSE;
				AxisStep 				:= STATE_WAIT;
				Axis3.cmdStop 			:= FALSE;
			ELSIF (Axis3.cmdManualForward  AND gMpAxisCoupling_3.Active) THEN
				gMpAxisCoupling_3.Cam 	:=TRUE;
				AxisStep := STATE_JOG;
			END_IF

			IF gMpAxisBasic_Axis3.Error THEN
				AxisStep := STATE_ERROR;
			END_IF

		STATE_STOP : //*********************** 11 ****************************** STATE_STOP ***************************** 11 ********************** STATE_STOP

			gMpAxisBasic_AxisVirtu3.Stop := TRUE;
			(* if axis is stopped go to state wait *)
			IF (gMpAxisBasic_AxisVirtu3.Stopped = 1  ) THEN
				gMpAxisBasic_AxisVirtu3.Stop := 0;
				AxisStep := STATE_READY;
			END_IF
			(* check if error occured *)
			IF (gMpAxisBasic_Axis3.Error ) THEN
				Axis3_ErrorID := 3;
				AxisStep := STATE_ERROR;
			END_IF

		STATE_JOG : //************************* 17 **************************** STATE_JOG ********************************* 17 ********************* STATE_JOG

			IF ( Axis3.cmdManualForward  AND gMpAxisCoupling_3.InSync) THEN
				gMpAxisBasic_AxisVirtu3.MoveAdditive:= TRUE;
			END_IF

			IF NOT(Axis3.cmdManualForward ) THEN
				gMpAxisBasic_AxisVirtu3.MoveAdditive:= FALSE;
				//				Axis1Home					:= FALSE;
				//				Axis2Home					:= FALSE;
				//				Axis3.cmdHome		 		:= FALSE;
				IF (NOT gMpAxisBasic_AxisVirtu3.CommandBusy AND NOT gMpAxisBasic_Axis3.CommandBusy) THEN
					AxisStep 				:= STATE_READY;
					//					gMpAxisCoupling_1.Enable	:= FALSE;
					//					gMpAxisCoupling_1.Cam 		:= FALSE;
				END_IF
				//				AxisStep := STATE_READY;
			END_IF

			(* check if error occured *)
			IF (gMpAxisBasic_Axis3.Error OR gMpAxisBasic_Axis3.Error) THEN
				Axis3_ErrorID := 4;
				AxisStep := STATE_ERROR;
			END_IF

		STATE_ERROR : //********************** 101 ******************************* STATE_ERROR **************************** 101 ********************** STATE_ERROR

			Axis3.statusStarting 		:=0;
			Axis3.statusFaulted 		:= TRUE;
			gMpAxisCoupling_3.Gear 		:= FALSE;
			gMpAxisCoupling_3.Cam 		:= FALSE;
			gMpAxisBasic_Axis3.Power 	:= FALSE;
			gMpAxisBasic_Axis3.Home 	:= FALSE;
			gMpAxisBasic_Axis3.Stop 	:= FALSE;
			gMpAxisBasic_AxisVirtu3.Power 		:= FALSE;
			gMpAxisBasic_AxisVirtu3.Home 		:= FALSE;
			gMpAxisBasic_AxisVirtu3.Stop 		:= FALSE;
			gMpAxisBasic_Axis3.MoveAbsolute 	:= FALSE;
			gMpAxisBasic_AxisVirtu3.MoveVelocity := FALSE;
			gMpAxisBasic_AxisVirtu3.MoveAbsolute := FALSE;
			gMpAxisBasic_AxisVirtu3.MoveVelocity := FALSE;
			gMpAxisBasic_Axis3.ErrorReset 		:= TRUE;
			gMpAxisBasic_AxisVirtu3.ErrorReset 	:= TRUE;
			gMpAxisCoupling_3.ErrorReset   		:= TRUE;

			IF (NOT(gMpAxisBasic_Axis3.Error ) AND NOT(gMpAxisBasic_AxisVirtu3.Error )) THEN
				Axis3.statusFaulted:=FALSE;
				gMpAxisBasic_Axis3.ErrorReset 		:= FALSE;
				gMpAxisBasic_AxisVirtu3.ErrorReset 	:= FALSE;
				gMpAxisCoupling_3.ErrorReset   		:= FALSE;
				AxisStep := STATE_WAIT;
				Axis3.statusErrorID := 0;
			END_IF

	END_CASE

	gMpAxisBasic_Axis3();
	gMpAxisBasic_Axis2();
	gMpAxisBasic_AxisVirtu3();
	gMpAxisCoupling_3();

	Axis3.cmdManualForward 	:= gActivateMotion;

END_PROGRAM
```

#### Exit.st
```iecst
PROGRAM _EXIT
	(* Insert code here *)
	gMpAxisBasic_Axis3.Enable 		:= FALSE;
	gMpAxisBasic_Axis3();
	gMpAxisBasic_AxisVirtu3.Enable 		:= TRUE;
	gMpAxisBasic_AxisVirtu3();
	gMpAxisCoupling_3.Enable			:= FALSE;
	gMpAxisCoupling_3();
END_PROGRAM
```

#### Init.st
```iecst
PROGRAM _INIT
	(* Insert code here *)
	Axis1.Exists := TRUE;
	gMpAxisBasicParType_AxisVirtu3.Position := 360.0;
	gMpAxisBasicParType_AxisVirtu3.Distance := 360.0;
	gMpAxisBasicParType_AxisVirtu3.Velocity := 360.0;
	gMpAxisBasicParType_AxisVirtu3.Deceleration := 1500;
	gMpAxisBasicParType_AxisVirtu3.Acceleration := 1500;
	gCouplingPar3.Cam.MasterScaling := 36000;
	gCouplingPar3.Cam.SlaveScaling := 36000;

END_PROGRAM
```

- Data object Logical/Cam3 (Cam) - Cam - Lift Speed Automat (no source held here)

### Program Logical/LDMPAccess (IEC)

#### Variables.var
```iecst
VAR
	MpAxisBasic_0 : MpAxisBasic;
END_VAR
```

#### Cyclic.ld
Ladder, written as Structured Text:
```iecst
PROGRAM _CYCLIC
END_PROGRAM
```

#### Exit.ld
Ladder, written as Structured Text:
```iecst
PROGRAM _EXIT
END_PROGRAM
```

Listed in the project but not available here: Logical/MNG_Global.typ, Logical/Libraries/ComTCP, Logical/Images
